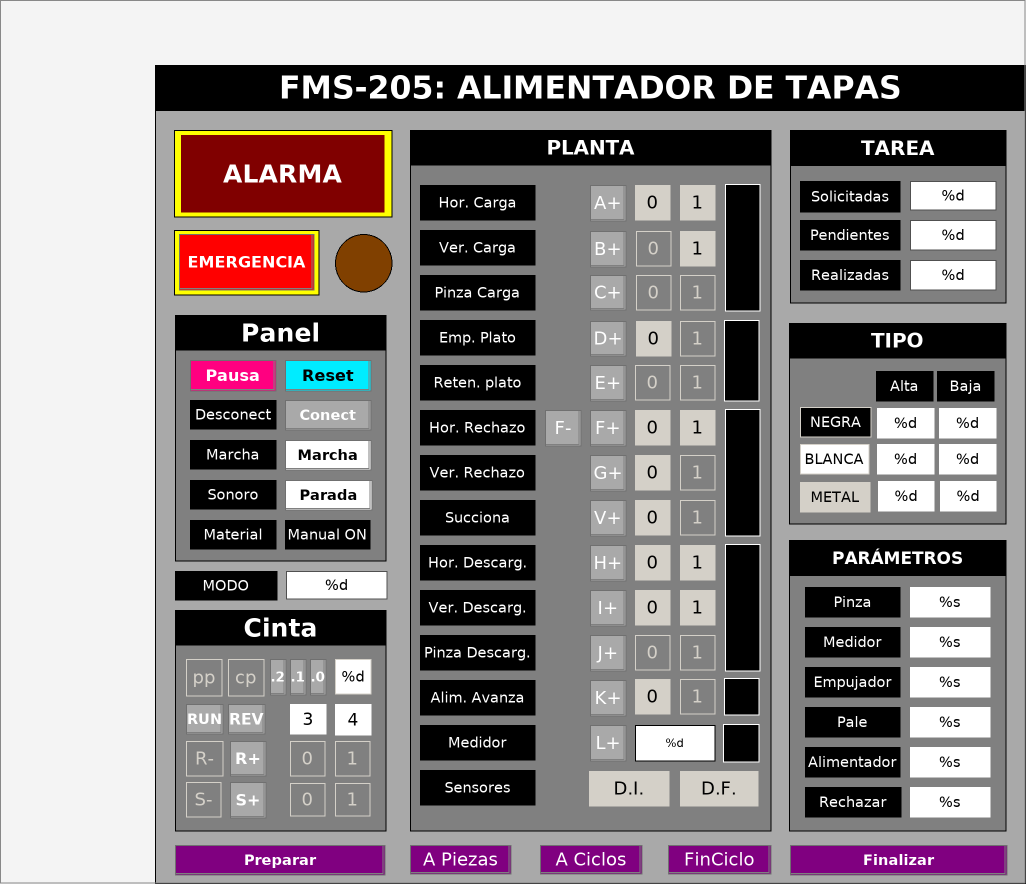
VISUALIZATION Visualization  // 1026x884
    Rectangle (155,110 871x774)
    Rectangle (175,315 211x246)
    Rectangle (410,160 361x671)
    Rectangle (420,185 115x35), "Hor. Carga"
    Rectangle (420,230 115x35), "Ver. Carga"
        toggle MAIN.Estacion.CargadorCierra
    Rectangle (420,275 115x35), "Pinza Carga"
    Rectangle (420,320 115x35), "Emp. Plato"
    Rectangle (420,365 115x35), "Reten. plato"
    Rectangle (420,410 115x35), "Hor. Rechazo"
    Rectangle (420,680 115x35), "Alim. Avanza"
    Rectangle (420,455 115x35), "Ver. Rechazo"
    Rectangle (420,500 115x35), "Succiona"
    Rectangle (420,545 115x35), "Hor. Descarg."
    Rectangle (420,590 115x35), "Ver. Descarg."
    Rectangle (420,635 115x35), "Pinza Descarg."
    Rectangle (420,725 115x35), "Medidor"
    Button (590,185 36x36), "A+", colour toggle: MAIN.Estacion.CargadorAvanza
        toggle MAIN.Estacion.CargadorAvanza
    Button (590,231 36x36), "B+", colour toggle: MAIN.Estacion.CargadorBaja
        toggle MAIN.Estacion.CargadorBaja
    Button (590,275 36x35), "C+", colour toggle: MAIN.Estacion.CargadorCierra
        toggle MAIN.Estacion.CargadorCierra
    Button (590,321 36x35), "D+", colour toggle: MAIN.Estacion.PlatoEmpujadorAvanza
        toggle MAIN.Estacion.PlatoEmpujadorAvanza
    Button (590,545 36x36), "H+", colour toggle: MAIN.Estacion.DescargadorAvanza
        toggle MAIN.Estacion.DescargadorAvanza
    Button (590,365 36x36), "E+", colour toggle: MAIN.Estacion.PlatoRetenedorAtras
        toggle MAIN.Estacion.PlatoRetenedorAtras
    Button (590,410 36x36), "F+", colour toggle: MAIN.Estacion.RechazadorAvanza
        toggle MAIN.Estacion.RechazadorAvanza
    Button (590,455 36x36), "G+", colour toggle: MAIN.Estacion.RechazadorBaja
        toggle MAIN.Estacion.RechazadorBaja
    Button (545,410 36x36), "F-", colour toggle: MAIN.Estacion.RechazadorRetrocede
        toggle MAIN.Estacion.RechazadorRetrocede
    Button (590,590 36x36), "I+", colour toggle: MAIN.Estacion.DescargadorAbajo
        toggle MAIN.Estacion.DescargadorAbajo
    Button (590,500 36x36), "V+", colour toggle: MAIN.Estacion.RechazadorSucciona
        toggle MAIN.Estacion.RechazadorSucciona
    Button (590,635 36x36), "J+", colour toggle: MAIN.Estacion.DescargadorCierra
        toggle MAIN.Estacion.DescargadorCierra
    Button (590,725 36x36), "L+", colour toggle: MAIN.Estacion.MedidorBaja
        toggle MAIN.Estacion.MedidorBaja
    Rectangle (410,130 361x35), "PLANTA"
    Button (285,440 86x30), "Marcha", colour toggle: MAIN.Estacion.PulsadorMarcha
        tap MAIN.Estacion.PulsadorMarcha
        toggle MAIN.Estacion.PulsadorMarcha
    Button (285,400 86x30), "Conect", colour toggle: MAIN.Estacion.EstacionConectada
        toggle MAIN.Estacion.EstacionConectada
    Rectangle (175,315 211x35), "Panel"
    Rectangle (789,323 217x201)
    Rectangle (789,323 217x35), "TIPO"
    Rectangle (175,620 211x211)
    Button (186,704 37x30), "RUN", colour toggle: MAIN.Estacion.CintaActiva
        toggle MAIN.Estacion.CintaActiva
    Button (228,704 37x30), "REV", colour toggle: MAIN.Estacion.CintaInvierte
        toggle MAIN.Estacion.CintaInvierte
    Rectangle (175,610 211x35), "Cinta"
    Rectangle (420,770 115x35), "Sensores"
    Rectangle (155,65 871x45), "FMS-205: ALIMENTADOR DE TAPAS"
    Rectangle (635,185 35x35), "0", colour toggle: MAIN.Estacion.CargadorDetras
    Rectangle (680,185 35x35), "1", colour toggle: MAIN.Estacion.CargadorDelante
    Rectangle (725,184 35x127), colour toggle: MAIN.Estacion.CargarPieza.Execute
    Rectangle (636,231 35x35), "0", colour toggle: MAIN.Estacion.CargadorAbajo
    Rectangle (680,231 35x35), "1", colour toggle: MAIN.Estacion.CargadorArriba
    Rectangle (636,275 35x35), "0"
    Rectangle (680,275 35x35), "1"
    Rectangle (635,410 35x35), "0", colour toggle: MAIN.Estacion.RechazadorDetras
    Rectangle (636,321 35x35), "0", colour toggle: MAIN.Estacion.PlatoEmpujadorDetras
    Rectangle (680,321 35x35), "1"
    Rectangle (724,320 35x81), colour toggle: MAIN.Estacion.EmpujarPlato.Execute
    Rectangle (635,365 35x35), "0"
    Rectangle (680,365 35x35), "1"
    Rectangle (680,410 35x35), "1", colour toggle: MAIN.Estacion.RechazadorDelante
    Rectangle (725,409 35x127), colour toggle: MAIN.Estacion.RechazarPieza.Execute
    Rectangle (635,545 35x35), "0", colour toggle: MAIN.Estacion.DescargadorDetras
    Rectangle (635,455 35x35), "0", colour toggle: MAIN.Estacion.RechazadorArriba
    Rectangle (680,455 35x35), "1"
    Rectangle (635,500 35x35), "0", colour toggle: MAIN.Estacion.RechazadorVacio
    Rectangle (680,500 35x35), "1"
    Rectangle (680,545 35x35), "1", colour toggle: MAIN.Estacion.DescargadorDelante
    Rectangle (725,544 35x127), colour toggle: MAIN.Estacion.DescargarPieza.Execute
    Rectangle (635,679 35x35), "0", colour toggle: MAIN.Estacion.AlimentadorDelante
    Rectangle (635,590 35x35), "0", colour toggle: MAIN.Estacion.DescargadorAbajo
    Rectangle (680,590 35x35), "1", colour toggle: MAIN.Estacion.DescargadorArriba
    Rectangle (635,635 35x35), "0"
    Rectangle (680,635 35x35), "1"
    Rectangle (680,679 35x35), "1"
    Rectangle (724,678 35x37), colour toggle: MAIN.Estacion.AvanzarAlimentador.Execute
    Rectangle (723,724 36x38), colour toggle: MAIN.Estacion.Medir.Execute
    Button (230,741 36x35), "R+", colour toggle: MAIN.Estacion.RetenedorBaja
        toggle MAIN.Estacion.RetenedorBaja
    Button (230,782 36x36), "S+"
        toggle MAIN.Estacion.SeparadorSube
    Button (270,659 16x36), ".2", colour toggle: MAIN.Estacion.CodigoPaleBit2
        toggle MAIN.Estacion.CodigoPaleBit2
    Button (290,659 16x36), ".1", colour toggle: MAIN.Estacion.CodigoPaleBit1
        toggle MAIN.Estacion.CodigoPaleBit1
    Button (310,659 16x36), ".0", colour toggle: MAIN.Estacion.CodigoPaleBit0
        toggle MAIN.Estacion.CodigoPaleBit0
    Rectangle (290,741 35x35), "0"
    Rectangle (335,741 35x35), "1"
    Rectangle (290,783 35x33), "0"
    Rectangle (335,783 35x33), "1"
    Rectangle (186,741 37x35), "R-"
    Rectangle (186,782 35x35), "S-"
    Rectangle (285,520 85x29), "Manual ON", colour toggle: MAIN.Estacion.SelectorManual
    Button (285,480 87x30), "Parada", colour toggle: MAIN.Estacion.PulsadorParada
        toggle MAIN.Estacion.PulsadorParada
    Rectangle (190,520 86x29), "Material", colour toggle: MAIN.Estacion.LamparaMaterial
    Button (590,680 36x36), "K+", colour toggle: MAIN.Estacion.AlimentadorAvanza
        toggle MAIN.Estacion.AlimentadorAvanza
    Rectangle (635,725 80x36), "%d", text variable: MAIN.Estacion.Codificador
    Rectangle (290,704 36x30), "3", colour toggle: MAIN.Estacion.CintaActiva AND MAIN.Estacion.CintaInvierte
    Rectangle (335,704 36x31), "4", colour toggle: MAIN.Estacion.CintaActiva AND NOT MAIN.Estacion.CintaInvierte
    Rectangle (789,540 217x36), "PARÁMETROS"
    Rectangle (789,575 217x256)
    RoundedRectangle (805,667 95x30), "Empujador"
    RoundedRectangle (805,707 95x30), "Pale"
    RoundedRectangle (805,747 95x30), "Alimentador"
    RoundedRectangle (805,787 96x30), "Rechazar"
    Rectangle (910,667 80x30), "%s", text variable: MAIN.Estacion.TpoEmpujadorAvanza
        OnMouseClick: write the text variable via Default
    Rectangle (910,707 80x30), "%s", text variable: MAIN.Estacion.TpoPaleEntrada
        OnMouseClick: write the text variable via Default
    Rectangle (910,747 80x30), "%s", text variable: MAIN.Estacion.TpoAlimentador
        OnMouseClick: write the text variable via Default
    Rectangle (910,787 80x30), "%s", text variable: MAIN.Estacion.TpoRechazador
        OnMouseClick: write the text variable via Default
    RoundedRectangle (805,627 95x30), "Medidor"
    RoundedRectangle (805,587 95x30), "Pinza"
    Rectangle (910,587 80x30), "%s", text variable: MAIN.Estacion.TpoPinza
        OnMouseClick: write the text variable via Default
    Rectangle (910,627 80x30), "%s", text variable: MAIN.Estacion.TpoMedidor
        OnMouseClick: write the text variable via Default
    Rectangle (790,130 216x36), "TAREA"
    Rectangle (790,165 216x138)
    RoundedRectangle (800,181 100x31), "Solicitadas"
    Rectangle (910,181 86x29), "%d", text variable: MAIN.Estacion.UnidadesSolicitadas
        OnMouseClick: write the text variable via Default
    RoundedRectangle (800,220 100x30), "Pendientes"
    Rectangle (910,220 86x30), "%d", text variable: MAIN.Estacion.UnidadesPendientes
        OnMouseClick: write the text variable via Default
    RoundedRectangle (800,260 100x30), "Realizadas"
    Rectangle (910,260 86x30), "%d", text variable: MAIN.Estacion.UnidadesRealizadas
        OnMouseClick: write the text variable via Default
    Rectangle (877,408 57x30), "%d", text variable: MAIN.Estacion.ListaPiezasSolicitadas[1]
        OnMouseClick: write the text variable via Default
    Rectangle (877,444 57x30), "%d", text variable: MAIN.Estacion.ListaPiezasSolicitadas[2]
        OnMouseClick: write the text variable via Default
    Rectangle (878,481 56x30), "%d", text variable: MAIN.Estacion.ListaPiezasSolicitadas[3]
        OnMouseClick: write the text variable via Default
    Button (540,845 102x29), "A Ciclos", colour toggle: MAIN.Estacion.CicloACiclo
        toggle MAIN.Estacion.CicloACiclo
    Button (190,360 86x31), "Pausa", colour toggle: MAIN.Estacion.PausaEstado
        toggle MAIN.Estacion.PausaEstado
    Button (285,360 86x31), "Reset", colour toggle: MAIN.Estacion.ReiniciaEstado
        tap MAIN.Estacion.ReiniciaEstado
    Rectangle (335,659 36x35), "%d", text variable: MAIN.Estacion.CodigoPale
    Rectangle (589,771 80x35), "D.I.", colour toggle: MAIN.Estacion.DetectorInductivo
    Rectangle (680,771 78x35), "D.F.", colour toggle: MAIN.Estacion.DetectorFotoelectrico
    RoundedRectangle (800,407 71x30), "NEGRA"
    RoundedRectangle (800,444 69x30), "BLANCA"
    RoundedRectangle (800,482 70x30), "METAL"
    RoundedRectangle (876,371 57x30), "Alta"
    RoundedRectangle (937,371 57x30), "Baja"
    Rectangle (939,408 57x30), "%d", text variable: MAIN.Estacion.ListaPiezasSolicitadas[4]
        OnMouseClick: write the text variable via Default
    Rectangle (939,444 57x30), "%d", text variable: MAIN.Estacion.ListaPiezasSolicitadas[5]
        OnMouseClick: write the text variable via Default
    Rectangle (940,481 56x30), "%d", text variable: MAIN.Estacion.ListaPiezasSolicitadas[6]
        OnMouseClick: write the text variable via Default
    Rectangle (186,659 36x37), "pp", text variable: MAIN.Estacion.PresenciaPale
    Rectangle (228,659 36x37), "cp"
    Rectangle (190,440 86x29), "Marcha", colour toggle: MAIN.Estacion.LamparaMarcha
    Rectangle (190,400 86x29), "Desconect", colour toggle: MAIN.Estacion.DesconectaEstacion
    Rectangle (190,480 86x29), "Sonoro", colour toggle: MAIN.Estacion.AvisadorSonoro
    Rectangle (174,130 218x87)
    Rectangle (180,134 205x79), "ALARMA", colour toggle: MAIN.Estacion.LamparaAlarma
    Rectangle (174,230 145x65)
    Button (179,234 135x56), "EMERGENCIA", colour toggle: MAIN.Estacion.PulsadorEmergencia
        toggle MAIN.Estacion.PulsadorEmergencia
    Rectangle (286,571 101x28), "%d", text variable: MAIN.Estacion.Director.Modo
        OnMouseClick: write the text variable via Default
    Rectangle (175,571 102x29), "MODO"
    Button (668,845 103x29), "FinCiclo", colour toggle: MAIN.Estacion.FinCiclo
        toggle MAIN.Estacion.FinCiclo
    Button (175,845 210x30), "Preparar", colour toggle: MAIN.Estacion.PrepararProduccion
        toggle MAIN.Estacion.PrepararProduccion
    Button (790,845 217x30), "Finalizar", colour toggle: MAIN.Estacion.FinalizarProduccion
        toggle MAIN.Estacion.FinalizarProduccion
    Ellipse (335,234 57x58), colour toggle: MAIN.Estacion.Director.Defecto
    Button (410,845 101x29), "A Piezas", colour toggle: MAIN.Estacion.PiezaAPieza
        toggle MAIN.Estacion.PiezaAPieza
END_VISUALIZATION

(* stored: Version 1.1.0.1, ProductVersion 3.1.4024.12
   Visu Visualization: Id {b02782e5-7dad-4791-9534-907cf86a8d7d} *)
